FUNCTION_BLOCK FB_StorageBypassGrnDivertTC
VAR_INPUT
	
	pCmp: POINTER TO CmpConvDivert;

END_VAR

VAR
	
	MainRunning: BOOL;
	SpurRunning: BOOL;
	
	onsPuckReady: R_TRIG;
	ResolvedDBStatusRouteGreen: cResolvedDBStatusRoute;
	ResolvedDBStatusRouteRed: cResolvedDBStatusRoute;
	ResolvedDBStatusRouteBlue: cResolvedDBStatusRoute;
	DBRouteToMain: BOOL;
	RouteToSpur: BOOL;
	
	
	tmrSpurNotOKToReceive: TON;
	
	Debug_DivertAllToMain: BOOL;
	Debug_DivertAllToSpur: BOOL;
	
END_VAR

// Traffic control for specific dirvert - Stn060
// 
// Currently each divert has independent/unique function block as it is expected that they will
//   eventually need to be tweeked for specific application

// Sum of main/spur running conditions... don't release if not running
MainRunning :=
	pCmp^.MainHeartbeatOK AND
	pCmp^.MainConvRunning;

SpurRunning :=
	pCmp^.SpurHeartbeatOK AND
	pCmp^.SpurConvRunning;


// On rising edege of puck ready interperate the puck/device data to see if it should be diverted to spur
onsPuckReady(CLK:=pCmp^.PuckReady);
IF onsPuckReady.Q THEN 	
	// Call function to turn DB puck/device status/route into single readable resolution
	ResolvedDBStatusRouteGreen :=
		FN_ResolveDBStatusRoutePuck(
			Puck := pCmp^.Puck,
			RouteToWork := cDBDetailRoute.TrayLoadGreen);
	ResolvedDBStatusRouteRed :=
		FN_ResolveDBStatusRoutePuck(
			Puck := pCmp^.Puck,
			RouteToWork := cDBDetailRoute.TrayLoadRed);
	ResolvedDBStatusRouteBlue :=
		FN_ResolveDBStatusRoutePuck(
			Puck := pCmp^.Puck,
			RouteToWork := cDBDetailRoute.TrayLoadBlue);
		
	// Use DB route and other possible line status to determine if puck should go to spur
	// This station never works on an empty puck.
	
	DBRouteToMain := 
		(ResolvedDBStatusRouteGreen = cResolvedDBStatusRoute.Normal_RoutedThisStation OR 
		ResolvedDBStatusRouteRed = cResolvedDBStatusRoute.Normal_RoutedThisStation OR
		ResolvedDBStatusRouteBlue = cResolvedDBStatusRoute.Normal_RoutedThisStation);
	
END_IF

RouteToSpur := NOT DBRouteToMain;
	
// Run timer for spur not ok to receive
// TODO - RCC: Eventualy include upstream buffer full before forcing release
tmrSpurNotOKToReceive(
		IN:= NOT SpurRunning OR NOT pCmp^.senSpurBufferFullOff,
		PT:= T#1000MS);
		
// Release main if that is DB route or if spur not ready in time
//  and a few other misc conditions.
//if main BF, release ALL to spur.

//pCmp^.MainBufferFull := NOT pCmp^.senMainBufferFullOff;

pCmp^.PuckReleaseMain := 
	pCmp^.PuckReady AND
	MainRunning AND
	(DBRouteToMain OR
//	tmrSpurNotOkToReceive.Q OR
	pCmp^.UnknownPuck OR
	Debug_DivertAllToMain) AND
	NOT Debug_DivertAllToSpur AND
	pCmp^.senMainBufferFullOff;
	
// Release to spur if that is route and it is available.
pCmp^.PuckReleaseSpur :=
	pCmp^.PuckReady AND
	MainRunning AND
	SpurRunning AND
	((RouteToSpur AND
	NOT pCmp^.UnknownPuck) OR
	Debug_DivertAllToSpur) AND
	NOT Debug_DivertAllToMain OR
	NOT pCmp^.senMainBufferFullOff;

END_FUNCTION_BLOCK

(* stored: Version 1.1.0.1, ProductVersion 3.1.4024.6
   POU FB_StorageBypassGrnDivertTC: Id {4970358b-0a02-4942-9c9a-7e78a74f739f}, SpecialFunc None *)
